TYPE ST_Floor :
STRUCT
	Call :BOOL;
	High,
	Mid,
	Low :BOOL;
END_STRUCT
END_TYPE

(* stored: Version 1.1.0.1, ProductVersion 3.1.4024.11
   DUT ST_Floor: Id {e7c47cb4-bc9a-451f-ad61-a0d5dc4b8f0f} *)
